	        #instOutputControlCathodeAlignSuctionOff(Enable := #statNowCmd = #STAT_LOOP,
	                                                 Condition1 := #instOutputCamCathodePnPX2Bwd.CamOutput,
	                                                 Condition2 := #instOutputCamCathodePnPZ2Down1.CamOutput,
	                                                 Condition3 := #instOutputCamCathodeAlignSuctionOff.CamOutput,
	                                                 Condition4 := #instOutputCamCathodePnPZ2Up1.CamOutput,
	                                                 Output := #statCathodeAlignSuction);

	        #instOutputControlCathodeAlignSuctionBlow(Enable := #statNowCmd = #STAT_LOOP,
	                                                  Condition1 := #instOutputCamCathodePnPX2Bwd.CamOutput,
	                                                  Condition2 := #instOutputCamCathodePnPZ2Down1.CamOutput,
	                                                  Condition3 := #instOutputCamCathodeAlignSuctionOff.CamOutput,
	                                                  Output => #statCathodeAlignBlow);
	    END_REGION

	    REGION CATHODE REELCUT DATA DELETE
	        #instOutputControlCathodeReelCutDataDeleteOn(Enable := #statNowCmd = #STAT_LOOP,
	                                                     Condition1 := #instOutputCamCathodePnPX1Bwd.CamOutput,
	                                                     Condition2 := #instOutputCamCathodePnPZ1Down1.CamOutput,
	                                                     Condition3 := #instOutputCamCathodePnPZ1ReelCutDataDeleteOn.CamOutput,
	                                                     Condition4 := #instOutputCamCathodePnPX1Fwd.CamOutput,
	                                                     Output := #statCathodeReelCutDataDelete);

	        #instOutputControlCathodeReelCutDataDeleteOff(Enable := #statNowCmd = #STAT_LOOP,
	                                                      Condition1 := #instOutputCamCathodePnPX1Fwd.CamOutput,
	                                                      Condition2 := #instOutputCamCathodePnPX1ReelCutDataDeleteOff.CamOutput,
	                                                      Condition3 := #instOutputCamCathodePnPZ1Down2.CamOutput,
	                                                      Output := #statCathodeReelCutDataDelete);

	    END_REGION

	    REGION CATHODE ALIGN TABLE VISION
	        #instOutputControlCathodeAlignVision(Enable := #statNowCmd = #STAT_LOOP,
	                                           Condition1 := #instOutputCamCathodePnPX1Fwd.CamOutput,
	                                           Condition2 := #instOutputCamCathodePnPZ1Down2.CamOutput,
	                                           Condition3 := #instOutputCamCathodePnPZ1AlignVision.CamOutput,
	                                           Output => #statCathodeAlignVision);


	    END_REGION

	END_REGION

	REGION SIGNAL RESET
	    IF NOT #Execute THEN
	        #statAnodePnP1Suction := FALSE;
	        #statAnodePnP1Blow := FALSE;
	        #statAnodePnP1ReelCutBlow := FALSE;
	        #statAnodePnP2Suction := FALSE;
	        #statAnodePnP2Blow := FALSE;
	        #statAnodeAlignSuction := FALSE;
	        #statAnodeAlignBlow := FALSE;
	        #statAnodePnP1RotaryWork := FALSE;
	        #statAnodePnP1RotaryHome := FALSE;
	        #statAnodeReelCutDataDelete := FALSE;
	        #statAnodeAlignVision := FALSE;
	        #statCathodePnP1Suction := FALSE;
	        #statCathodePnP1Blow := FALSE;
	        #statCathodePnP1ReelCutBlow := FALSE;
	        #statCathodePnP2Suction := FALSE;
	        #statCathodePnP2Blow := FALSE;
	        #statCathodeAlignSuction := FALSE;
	        #statCathodeAlignBlow := FALSE;
	        #statCathodePnP1RotaryWork := FALSE;
	        #statCathodePnP1RotaryHome := FALSE;
	        #statCathodeReelCutDataDelete := FALSE;
	        #statCathodeAlignVision := FALSE;
	        #statStackTableZAnodeDown := FALSE;
	        #statStackTableZCathodeDown := FALSE;
	        #statStackAnodeVision := FALSE;
	        #statStackCathodeVision := FALSE;
	    END_IF;
	END_REGION

	REGION OUTPUT SIGNAL                                                            // 각 커맨드 동작 시 상태 표시 출력
	    #Output.AnodePnP1Suction := #statAnodePnP1Suction;
	    #Output.AnodePnP1Blow := #statAnodePnP1Blow;
	    #Output.AnodePnP1ReelCutBlow := #statAnodePnP1ReelCutBlow;
	    #Output.AnodePnP2Suction := #statAnodePnP2Suction;
	    #Output.AnodePnP2Blow := #statAnodePnP2Blow;
	    #Output.AnodeAlignSuction := #statAnodeAlignSuction;
	    #Output.AnodeAlignBlow := #statAnodeAlignBlow;
	    #Output.AnodePnP1RotaryWork := #statAnodePnP1RotaryWork;
	    #Output.AnodePnP1RotaryHome := #statAnodePnP1RotaryHome;
	    #Output.AnodeReelCutDataDelete := #statAnodeReelCutDataDelete;
	    #Output.AnodeAlignVision := #statAnodeAlignVision;
	    #Output.CathodePnP1Suction := #statCathodePnP1Suction;
	    #Output.CathodePnP1Blow := #statCathodePnP1Blow;
	    #Output.CathodePnP1ReelCutBlow := #statCathodePnP1ReelCutBlow;
	    #Output.CathodePnP2Suction := #statCathodePnP2Suction;
	    #Output.CathodePnP2Blow := #statCathodePnP2Blow;
	    #Output.CathodeAlignSuction := #statCathodeAlignSuction;
	    #Output.CathodeAlignBlow := #statCathodeAlignBlow;
	    #Output.CathodePnP1RotaryWork := #statCathodePnP1RotaryWork;
	    #Output.CathodePnP1RotaryHome := #statCathodePnP1RotaryHome;
	    #Output.CathodeReelCutDataDelete := #statCathodeReelCutDataDelete;
	    #Output.CathodeAlignVision := #statCathodeAlignVision;
	    #Output.StackTableZAnodeDown := #statStackTableZAnodeDown;
	    #Output.StackTableZCathodeDown := #statStackTableZCathodeDown;
	    #Output.StackAnodeVision := #statStackAnodeVision;
	    #Output.StackCathodeVision := #statStackCathodeVision;

	    #Busy := #statNowCmd = #STAT_START
	    OR #statNowCmd = #STAT_LOOP;
	    #Done := #statNowCmd = #STAT_DONE;
	    #Error := #statNowCmd = #STAT_ERROR;
	    #NowCmd := #statNowCmd;
	    #BeforeCmd := #statBeforeCmd;
	END_REGION
END_FUNCTION_BLOCK

